{attribute 'enable_dynamic_creation'}
FUNCTION_BLOCK FutureMCPower EXTENDS FB_AbstructFuture
VAR_INPUT
END_VAR
VAR_OUTPUT
END_VAR
VAR
	_axis: REFERENCE TO AXIS_REF;
	_override: LREAL := 100.0;
	_enable_positive:	BOOL := TRUE; 
	_enable_negative:	BOOL := TRUE;
	_fb_power	: MC_Power;
	_mc_reset	: MC_Reset;
	_mc_stop	: MC_Stop;
	_option : ST_PowerOptions;
	_buffer_mode : MC_BufferMode;
	_status : BOOL;
END_VAR

METHOD error_reset : BOOL // Must be overrided if future has any errors.
VAR_INST
	_exec_state : UDINT;
END_VAR
IF _error_id <> 0 THEN
	CASE _exec_state OF
		0:
			_mc_reset(Axis := _axis, Execute := FALSE);
			_mc_reset(Axis:= _axis, Execute := TRUE );
			_exec_state := 1;
		1:
			IF _mc_reset.Busy THEN
				_mc_reset(Axis:= _axis,Execute := FALSE);
				error_reset := TRUE;
			END_IF
	END_CASE	
	_error_id := _fb_power.ErrorID;
ELSE
	error_reset := TRUE;
END_IF
END_METHOD

METHOD execute : BOOL // Return TRUE if finish.
VAR_INST
	_exec_state: UINT;
	_stoped : BOOL;
END_VAR
_axis.ReadStatus();
IF _axis.Status.Moving THEN
	_stoped := FALSE;
	_exec_state := 0;
END_IF

IF NOT _stoped THEN
	CASE _exec_state OF
		0:
			_mc_stop(axis := _axis, Execute := FALSE);
			_mc_stop(
				Axis:= _axis,
				Execute := TRUE
			);
			_exec_state := 1;
		1:
			IF _mc_stop.Busy THEN
				_mc_stop(Axis:= _axis,Execute := FALSE);
				_stoped := TRUE;
			END_IF
	END_CASE
END_IF
	
IF _axis.Status.NotMoving AND _stoped THEN
	_fb_power(
		Axis:= _axis, 
		Enable:= _status, 
		Enable_Positive:= _enable_positive, 
		Enable_Negative:= _enable_negative, 
		Override:= _override, 
		BufferMode:= _buffer_mode, 
		Options:= _option, 
	);
	_error_id := _fb_power.ErrorID;
	execute := _status = _fb_Power.Status;
END_IF
END_METHOD

METHOD set_options : BOOL
VAR_INPUT
	Enable_Positive:	BOOL; 
	Enable_Negative:	BOOL;
	Override:			LREAL := 100;
	buffer_mode : MC_BufferMode;
	option : ST_PowerOptions;
END_VAR
_override := Override;
_enable_positive := Enable_Positive;
_enable_negative := Enable_Negative;
_buffer_mode := buffer_mode;
_option := option;
END_METHOD

METHOD set_parameters : BOOL
VAR_INPUT
	axis : REFERENCE TO AXIS_REF;
	status : BOOL;
END_VAR
_axis REF= axis;
_status := status;
_enable_positive := status;
_enable_negative := status;
END_METHOD

END_FUNCTION_BLOCK

(* stored: Version 1.1.0.1, ProductVersion 3.1.4026.13
   POU FutureMCPower: Id {53bbc5ad-8cba-4d76-9354-ff6510473cd2}, SpecialFunc None
   Method error_reset: Id {fbfcfc82-515e-4f7c-ae99-279462150b8a}
   Method execute: Id {f127afa9-edb6-44ee-8a9c-b074dfb931e5}
   Method set_options: Id {93406fea-fe89-4d4b-b9dc-dafbd821cdd6}
   Method set_parameters: Id {c4fee9f1-f0d8-457c-bc4c-46597f9f2a6d} *)
